FUNCTION_BLOCK FB_Observer_UDINT EXTENDS FB_AbstractObserver
VAR
    _nVal:              UDINT;
END_VAR

METHOD FB_init : BOOL
VAR_INPUT
	bInitRetains : BOOL; // if TRUE, the retain variables are initialized (warm start / cold start)
	bInCopyCode : BOOL;  // if TRUE, the instance afterwards gets moved into the copy code (online change)
END_VAR
THIS^._nTypeClass := __SYSTEM.TYPE_CLASS.TYPE_UDINT;
THIS^._pVal := ADR(THIS^._nVal);
THIS^._nSize := SIZEOF(THIS^._nVal);
END_METHOD

PROPERTY nValue32 : UDINT
GET
nValue32 := THIS^._nVal;
END_GET
END_PROPERTY

END_FUNCTION_BLOCK

(* stored: Version 1.1.0.1, ProductVersion 3.1.4024.12
   POU FB_Observer_UDINT: Id {d6527244-cad8-4610-99ab-4505dafbdc58}, SpecialFunc None
   Method FB_init: Id {08b1ba03-fe54-0423-2357-76b36c37199a}
   Property nValue32: Id {e0166b47-d1da-4a6d-abe6-c8c5d19c4651}
   Get Get: Id {8d705986-af7a-40f7-8080-4c9f0e662ea5} *)
